// TIA Portal V17 export
// export: Created 2026-04-12T10:31:11.5882867Z, ExportSetting WithDefaults, DisplayName Totally Integrated Automation Portal, DisplayVersion V17 Update 4, DisplayName TIA Portal Openness, DisplayVersion V17 Update 4, DisplayName TIA Portal Version Control Interface, DisplayVersion V17, DisplayName SINAMICS Startdrive Advanced, DisplayVersion V17, DisplayName SINAMICS Startdrive G130, G150, S120, S150, SINAMICS MV, S210, DisplayVersion V17, DisplayName SINAMICS Startdrive G110M, G120, G120C, G120D, G120P, G115D, DisplayVersion V17, DisplayName STEP 7 Professional, DisplayVersion V17 Update 4, DisplayName STEP 7 Safety, DisplayVersion V17, DisplayName WinCC Advanced, DisplayVersion V17 Update 4
FUNCTION "PID参数控制" : Void   // FC6, LAD
{ S7_Optimized_Access := 'TRUE' }
VERSION : 0.1
// stored: AutoNumber true, IsIECCheckEnabled false, SetENOAutomatically false, UDAEnableTagReadback false
BEGIN

REGION Network 1: 采样时间
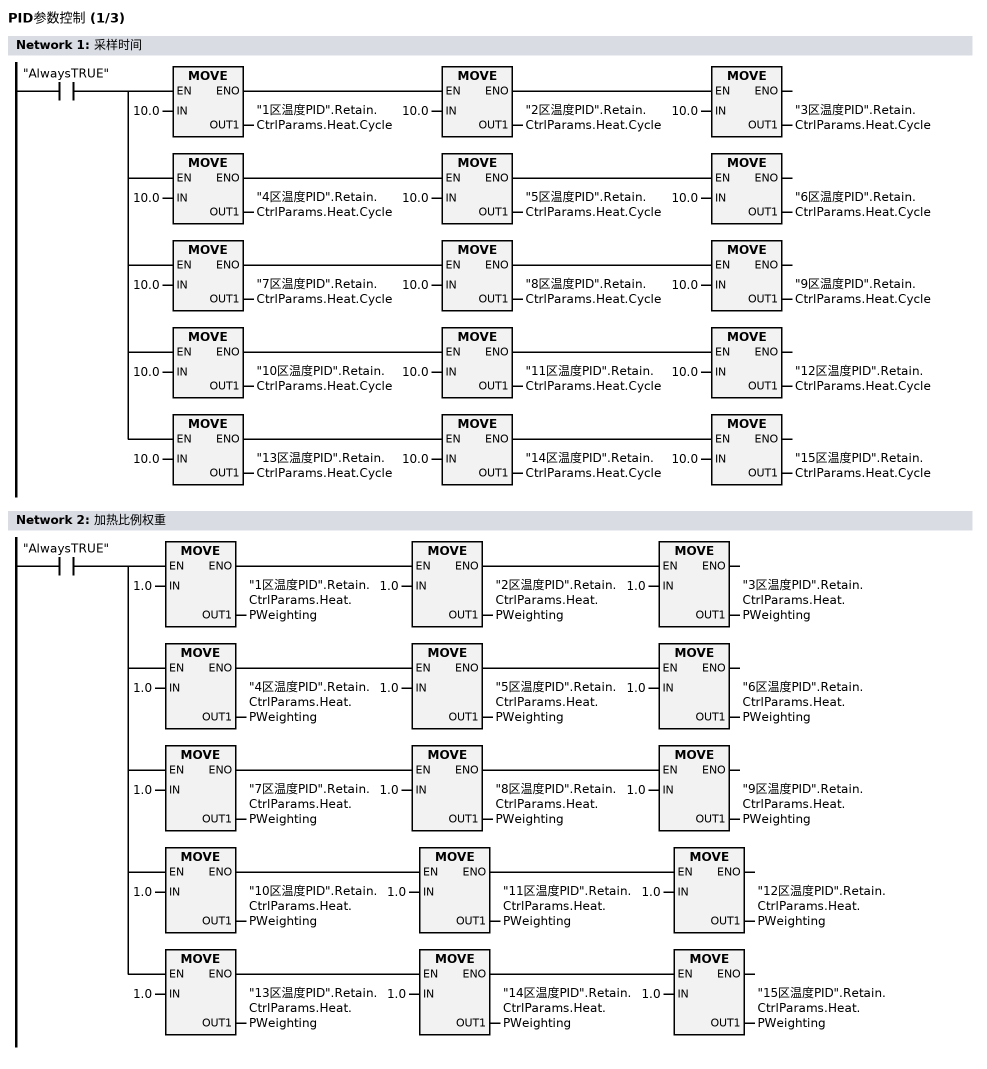
   RUNG wire#powerrail
      Contact( "AlwaysTRUE" )
      wire#w1
      Move(in := 10.0, out1 => "1区温度PID".Retain.CtrlParams.Heat.Cycle)
      Move(in := 10.0, out1 => "2区温度PID".Retain.CtrlParams.Heat.Cycle)
      Move(in := 10.0, out1 => "3区温度PID".Retain.CtrlParams.Heat.Cycle)
   END_RUNG
   RUNG wire#w1
      Move(in := 10.0, out1 => "4区温度PID".Retain.CtrlParams.Heat.Cycle)
      Move(in := 10.0, out1 => "5区温度PID".Retain.CtrlParams.Heat.Cycle)
      Move(in := 10.0, out1 => "6区温度PID".Retain.CtrlParams.Heat.Cycle)
   END_RUNG
   RUNG wire#w1
      Move(in := 10.0, out1 => "7区温度PID".Retain.CtrlParams.Heat.Cycle)
      Move(in := 10.0, out1 => "8区温度PID".Retain.CtrlParams.Heat.Cycle)
      Move(in := 10.0, out1 => "9区温度PID".Retain.CtrlParams.Heat.Cycle)
   END_RUNG
   RUNG wire#w1
      Move(in := 10.0, out1 => "10区温度PID".Retain.CtrlParams.Heat.Cycle)
      Move(in := 10.0, out1 => "11区温度PID".Retain.CtrlParams.Heat.Cycle)
      Move(in := 10.0, out1 => "12区温度PID".Retain.CtrlParams.Heat.Cycle)
   END_RUNG
   RUNG wire#w1
      Move(in := 10.0, out1 => "13区温度PID".Retain.CtrlParams.Heat.Cycle)
      Move(in := 10.0, out1 => "14区温度PID".Retain.CtrlParams.Heat.Cycle)
      Move(in := 10.0, out1 => "15区温度PID".Retain.CtrlParams.Heat.Cycle)
   END_RUNG
   // the same network as SCL:
   IF "AlwaysTRUE" THEN
       "1区温度PID".Retain.CtrlParams.Heat.Cycle := 10.0;
       "2区温度PID".Retain.CtrlParams.Heat.Cycle := 10.0;
       "3区温度PID".Retain.CtrlParams.Heat.Cycle := 10.0;
       "4区温度PID".Retain.CtrlParams.Heat.Cycle := 10.0;
       "5区温度PID".Retain.CtrlParams.Heat.Cycle := 10.0;
       "6区温度PID".Retain.CtrlParams.Heat.Cycle := 10.0;
       "7区温度PID".Retain.CtrlParams.Heat.Cycle := 10.0;
       "8区温度PID".Retain.CtrlParams.Heat.Cycle := 10.0;
       "9区温度PID".Retain.CtrlParams.Heat.Cycle := 10.0;
       "10区温度PID".Retain.CtrlParams.Heat.Cycle := 10.0;
       "11区温度PID".Retain.CtrlParams.Heat.Cycle := 10.0;
       "12区温度PID".Retain.CtrlParams.Heat.Cycle := 10.0;
       "13区温度PID".Retain.CtrlParams.Heat.Cycle := 10.0;
       "14区温度PID".Retain.CtrlParams.Heat.Cycle := 10.0;
       "15区温度PID".Retain.CtrlParams.Heat.Cycle := 10.0;
   END_IF;
END_REGION

REGION Network 2: 加热比例权重
   RUNG wire#powerrail
      Contact( "AlwaysTRUE" )
      wire#w1
      Move(in := 1.0, out1 => "1区温度PID".Retain.CtrlParams.Heat.PWeighting)
      Move(in := 1.0, out1 => "2区温度PID".Retain.CtrlParams.Heat.PWeighting)
      Move(in := 1.0, out1 => "3区温度PID".Retain.CtrlParams.Heat.PWeighting)
   END_RUNG
   RUNG wire#w1
      Move(in := 1.0, out1 => "4区温度PID".Retain.CtrlParams.Heat.PWeighting)
      Move(in := 1.0, out1 => "5区温度PID".Retain.CtrlParams.Heat.PWeighting)
      Move(in := 1.0, out1 => "6区温度PID".Retain.CtrlParams.Heat.PWeighting)
   END_RUNG
   RUNG wire#w1
      Move(in := 1.0, out1 => "7区温度PID".Retain.CtrlParams.Heat.PWeighting)
      Move(in := 1.0, out1 => "8区温度PID".Retain.CtrlParams.Heat.PWeighting)
      Move(in := 1.0, out1 => "9区温度PID".Retain.CtrlParams.Heat.PWeighting)
   END_RUNG
   RUNG wire#w1
      Move(in := 1.0, out1 => "10区温度PID".Retain.CtrlParams.Heat.PWeighting)
      Move(in := 1.0, out1 => "11区温度PID".Retain.CtrlParams.Heat.PWeighting)
      Move(in := 1.0, out1 => "12区温度PID".Retain.CtrlParams.Heat.PWeighting)
   END_RUNG
   RUNG wire#w1
      Move(in := 1.0, out1 => "13区温度PID".Retain.CtrlParams.Heat.PWeighting)
      Move(in := 1.0, out1 => "14区温度PID".Retain.CtrlParams.Heat.PWeighting)
      Move(in := 1.0, out1 => "15区温度PID".Retain.CtrlParams.Heat.PWeighting)
   END_RUNG
   // the same network as SCL:
   IF "AlwaysTRUE" THEN
       "1区温度PID".Retain.CtrlParams.Heat.PWeighting := 1.0;
       "2区温度PID".Retain.CtrlParams.Heat.PWeighting := 1.0;
       "3区温度PID".Retain.CtrlParams.Heat.PWeighting := 1.0;
       "4区温度PID".Retain.CtrlParams.Heat.PWeighting := 1.0;
       "5区温度PID".Retain.CtrlParams.Heat.PWeighting := 1.0;
       "6区温度PID".Retain.CtrlParams.Heat.PWeighting := 1.0;
       "7区温度PID".Retain.CtrlParams.Heat.PWeighting := 1.0;
       "8区温度PID".Retain.CtrlParams.Heat.PWeighting := 1.0;
       "9区温度PID".Retain.CtrlParams.Heat.PWeighting := 1.0;
       "10区温度PID".Retain.CtrlParams.Heat.PWeighting := 1.0;
       "11区温度PID".Retain.CtrlParams.Heat.PWeighting := 1.0;
       "12区温度PID".Retain.CtrlParams.Heat.PWeighting := 1.0;
       "13区温度PID".Retain.CtrlParams.Heat.PWeighting := 1.0;
       "14区温度PID".Retain.CtrlParams.Heat.PWeighting := 1.0;
       "15区温度PID".Retain.CtrlParams.Heat.PWeighting := 1.0;
   END_IF;
END_REGION

REGION Network 3: 微分比例权重
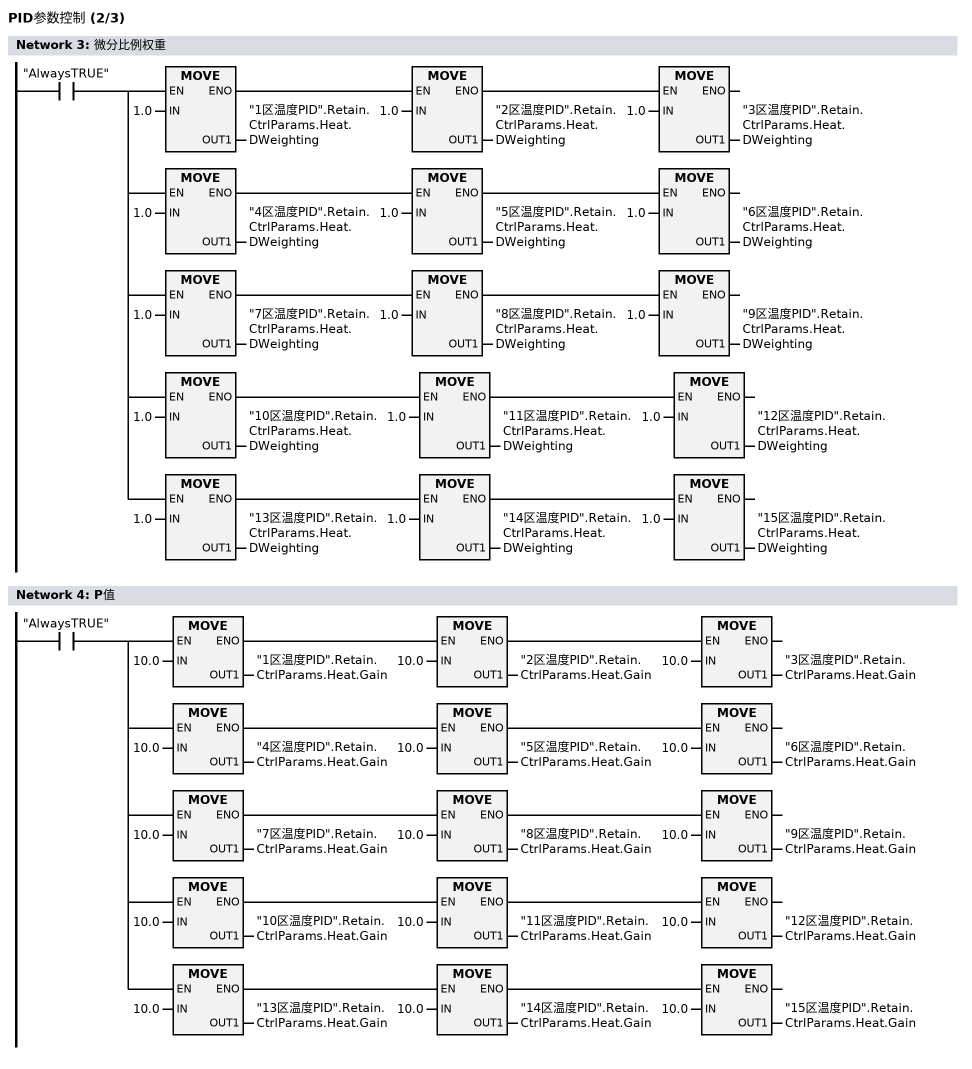
   RUNG wire#powerrail
      Contact( "AlwaysTRUE" )
      wire#w1
      Move(in := 1.0, out1 => "1区温度PID".Retain.CtrlParams.Heat.DWeighting)
      Move(in := 1.0, out1 => "2区温度PID".Retain.CtrlParams.Heat.DWeighting)
      Move(in := 1.0, out1 => "3区温度PID".Retain.CtrlParams.Heat.DWeighting)
   END_RUNG
   RUNG wire#w1
      Move(in := 1.0, out1 => "4区温度PID".Retain.CtrlParams.Heat.DWeighting)
      Move(in := 1.0, out1 => "5区温度PID".Retain.CtrlParams.Heat.DWeighting)
      Move(in := 1.0, out1 => "6区温度PID".Retain.CtrlParams.Heat.DWeighting)
   END_RUNG
   RUNG wire#w1
      Move(in := 1.0, out1 => "7区温度PID".Retain.CtrlParams.Heat.DWeighting)
      Move(in := 1.0, out1 => "8区温度PID".Retain.CtrlParams.Heat.DWeighting)
      Move(in := 1.0, out1 => "9区温度PID".Retain.CtrlParams.Heat.DWeighting)
   END_RUNG
   RUNG wire#w1
      Move(in := 1.0, out1 => "10区温度PID".Retain.CtrlParams.Heat.DWeighting)
      Move(in := 1.0, out1 => "11区温度PID".Retain.CtrlParams.Heat.DWeighting)
      Move(in := 1.0, out1 => "12区温度PID".Retain.CtrlParams.Heat.DWeighting)
   END_RUNG
   RUNG wire#w1
      Move(in := 1.0, out1 => "13区温度PID".Retain.CtrlParams.Heat.DWeighting)
      Move(in := 1.0, out1 => "14区温度PID".Retain.CtrlParams.Heat.DWeighting)
      Move(in := 1.0, out1 => "15区温度PID".Retain.CtrlParams.Heat.DWeighting)
   END_RUNG
   // the same network as SCL:
   IF "AlwaysTRUE" THEN
       "1区温度PID".Retain.CtrlParams.Heat.DWeighting := 1.0;
       "2区温度PID".Retain.CtrlParams.Heat.DWeighting := 1.0;
       "3区温度PID".Retain.CtrlParams.Heat.DWeighting := 1.0;
       "4区温度PID".Retain.CtrlParams.Heat.DWeighting := 1.0;
       "5区温度PID".Retain.CtrlParams.Heat.DWeighting := 1.0;
       "6区温度PID".Retain.CtrlParams.Heat.DWeighting := 1.0;
       "7区温度PID".Retain.CtrlParams.Heat.DWeighting := 1.0;
       "8区温度PID".Retain.CtrlParams.Heat.DWeighting := 1.0;
       "9区温度PID".Retain.CtrlParams.Heat.DWeighting := 1.0;
       "10区温度PID".Retain.CtrlParams.Heat.DWeighting := 1.0;
       "11区温度PID".Retain.CtrlParams.Heat.DWeighting := 1.0;
       "12区温度PID".Retain.CtrlParams.Heat.DWeighting := 1.0;
       "13区温度PID".Retain.CtrlParams.Heat.DWeighting := 1.0;
       "14区温度PID".Retain.CtrlParams.Heat.DWeighting := 1.0;
       "15区温度PID".Retain.CtrlParams.Heat.DWeighting := 1.0;
   END_IF;
END_REGION

REGION Network 4: P值
   RUNG wire#powerrail
      Contact( "AlwaysTRUE" )
      wire#w1
      Move(in := 10.0, out1 => "1区温度PID".Retain.CtrlParams.Heat.Gain)
      Move(in := 10.0, out1 => "2区温度PID".Retain.CtrlParams.Heat.Gain)
      Move(in := 10.0, out1 => "3区温度PID".Retain.CtrlParams.Heat.Gain)
   END_RUNG
   RUNG wire#w1
      Move(in := 10.0, out1 => "4区温度PID".Retain.CtrlParams.Heat.Gain)
      Move(in := 10.0, out1 => "5区温度PID".Retain.CtrlParams.Heat.Gain)
      Move(in := 10.0, out1 => "6区温度PID".Retain.CtrlParams.Heat.Gain)
   END_RUNG
   RUNG wire#w1
      Move(in := 10.0, out1 => "7区温度PID".Retain.CtrlParams.Heat.Gain)
      Move(in := 10.0, out1 => "8区温度PID".Retain.CtrlParams.Heat.Gain)
      Move(in := 10.0, out1 => "9区温度PID".Retain.CtrlParams.Heat.Gain)
   END_RUNG
   RUNG wire#w1
      Move(in := 10.0, out1 => "10区温度PID".Retain.CtrlParams.Heat.Gain)
      Move(in := 10.0, out1 => "11区温度PID".Retain.CtrlParams.Heat.Gain)
      Move(in := 10.0, out1 => "12区温度PID".Retain.CtrlParams.Heat.Gain)
   END_RUNG
   RUNG wire#w1
      Move(in := 10.0, out1 => "13区温度PID".Retain.CtrlParams.Heat.Gain)
      Move(in := 10.0, out1 => "14区温度PID".Retain.CtrlParams.Heat.Gain)
      Move(in := 10.0, out1 => "15区温度PID".Retain.CtrlParams.Heat.Gain)
   END_RUNG
   // the same network as SCL:
   IF "AlwaysTRUE" THEN
       "1区温度PID".Retain.CtrlParams.Heat.Gain := 10.0;
       "2区温度PID".Retain.CtrlParams.Heat.Gain := 10.0;
       "3区温度PID".Retain.CtrlParams.Heat.Gain := 10.0;
       "4区温度PID".Retain.CtrlParams.Heat.Gain := 10.0;
       "5区温度PID".Retain.CtrlParams.Heat.Gain := 10.0;
       "6区温度PID".Retain.CtrlParams.Heat.Gain := 10.0;
       "7区温度PID".Retain.CtrlParams.Heat.Gain := 10.0;
       "8区温度PID".Retain.CtrlParams.Heat.Gain := 10.0;
       "9区温度PID".Retain.CtrlParams.Heat.Gain := 10.0;
       "10区温度PID".Retain.CtrlParams.Heat.Gain := 10.0;
       "11区温度PID".Retain.CtrlParams.Heat.Gain := 10.0;
       "12区温度PID".Retain.CtrlParams.Heat.Gain := 10.0;
       "13区温度PID".Retain.CtrlParams.Heat.Gain := 10.0;
       "14区温度PID".Retain.CtrlParams.Heat.Gain := 10.0;
       "15区温度PID".Retain.CtrlParams.Heat.Gain := 10.0;
   END_IF;
END_REGION

REGION Network 5: I值
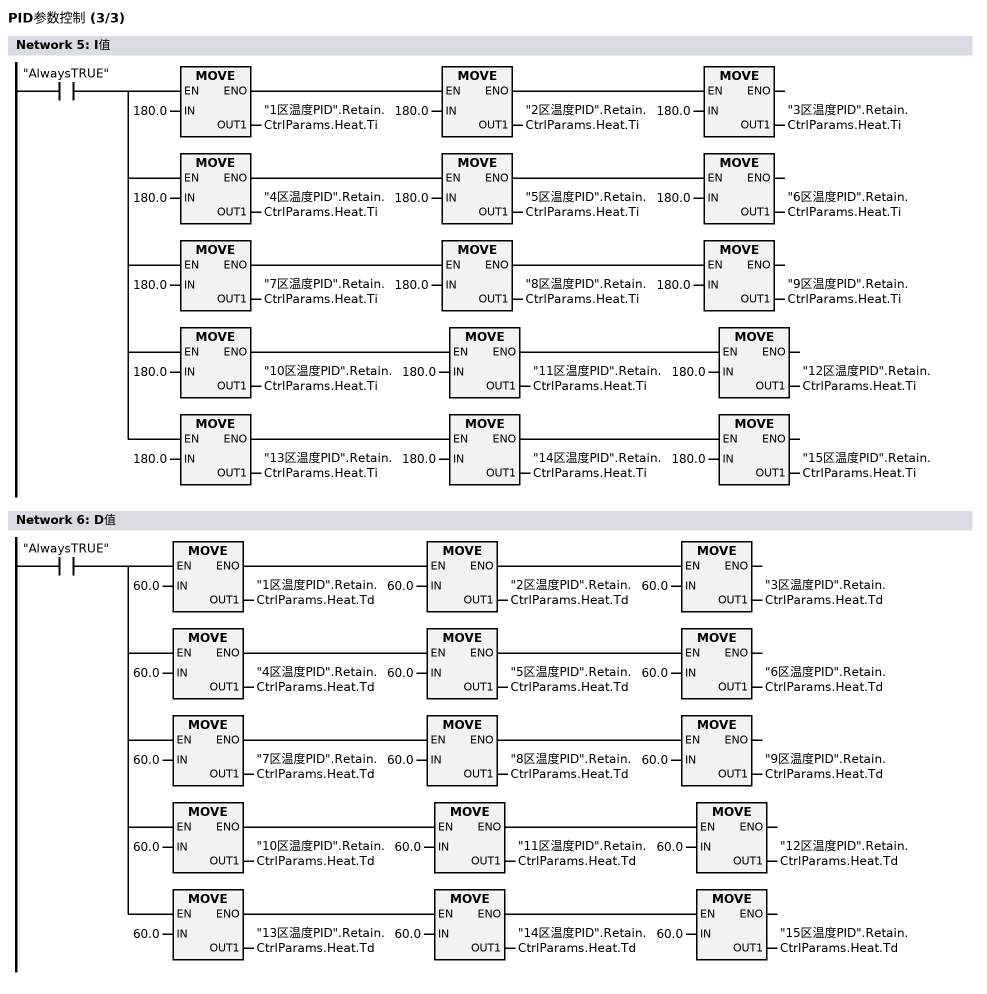
   RUNG wire#powerrail
      Contact( "AlwaysTRUE" )
      wire#w1
      Move(in := 180.0, out1 => "1区温度PID".Retain.CtrlParams.Heat.Ti)
      Move(in := 180.0, out1 => "2区温度PID".Retain.CtrlParams.Heat.Ti)
      Move(in := 180.0, out1 => "3区温度PID".Retain.CtrlParams.Heat.Ti)
   END_RUNG
   RUNG wire#w1
      Move(in := 180.0, out1 => "4区温度PID".Retain.CtrlParams.Heat.Ti)
      Move(in := 180.0, out1 => "5区温度PID".Retain.CtrlParams.Heat.Ti)
      Move(in := 180.0, out1 => "6区温度PID".Retain.CtrlParams.Heat.Ti)
   END_RUNG
   RUNG wire#w1
      Move(in := 180.0, out1 => "7区温度PID".Retain.CtrlParams.Heat.Ti)
      Move(in := 180.0, out1 => "8区温度PID".Retain.CtrlParams.Heat.Ti)
      Move(in := 180.0, out1 => "9区温度PID".Retain.CtrlParams.Heat.Ti)
   END_RUNG
   RUNG wire#w1
      Move(in := 180.0, out1 => "10区温度PID".Retain.CtrlParams.Heat.Ti)
      Move(in := 180.0, out1 => "11区温度PID".Retain.CtrlParams.Heat.Ti)
      Move(in := 180.0, out1 => "12区温度PID".Retain.CtrlParams.Heat.Ti)
   END_RUNG
   RUNG wire#w1
      Move(in := 180.0, out1 => "13区温度PID".Retain.CtrlParams.Heat.Ti)
      Move(in := 180.0, out1 => "14区温度PID".Retain.CtrlParams.Heat.Ti)
      Move(in := 180.0, out1 => "15区温度PID".Retain.CtrlParams.Heat.Ti)
   END_RUNG
   // the same network as SCL:
   IF "AlwaysTRUE" THEN
       "1区温度PID".Retain.CtrlParams.Heat.Ti := 180.0;
       "2区温度PID".Retain.CtrlParams.Heat.Ti := 180.0;
       "3区温度PID".Retain.CtrlParams.Heat.Ti := 180.0;
       "4区温度PID".Retain.CtrlParams.Heat.Ti := 180.0;
       "5区温度PID".Retain.CtrlParams.Heat.Ti := 180.0;
       "6区温度PID".Retain.CtrlParams.Heat.Ti := 180.0;
       "7区温度PID".Retain.CtrlParams.Heat.Ti := 180.0;
       "8区温度PID".Retain.CtrlParams.Heat.Ti := 180.0;
       "9区温度PID".Retain.CtrlParams.Heat.Ti := 180.0;
       "10区温度PID".Retain.CtrlParams.Heat.Ti := 180.0;
       "11区温度PID".Retain.CtrlParams.Heat.Ti := 180.0;
       "12区温度PID".Retain.CtrlParams.Heat.Ti := 180.0;
       "13区温度PID".Retain.CtrlParams.Heat.Ti := 180.0;
       "14区温度PID".Retain.CtrlParams.Heat.Ti := 180.0;
       "15区温度PID".Retain.CtrlParams.Heat.Ti := 180.0;
   END_IF;
END_REGION

REGION Network 6: D值
   RUNG wire#powerrail
      Contact( "AlwaysTRUE" )
      wire#w1
      Move(in := 60.0, out1 => "1区温度PID".Retain.CtrlParams.Heat.Td)
      Move(in := 60.0, out1 => "2区温度PID".Retain.CtrlParams.Heat.Td)
      Move(in := 60.0, out1 => "3区温度PID".Retain.CtrlParams.Heat.Td)
   END_RUNG
   RUNG wire#w1
      Move(in := 60.0, out1 => "4区温度PID".Retain.CtrlParams.Heat.Td)
      Move(in := 60.0, out1 => "5区温度PID".Retain.CtrlParams.Heat.Td)
      Move(in := 60.0, out1 => "6区温度PID".Retain.CtrlParams.Heat.Td)
   END_RUNG
   RUNG wire#w1
      Move(in := 60.0, out1 => "7区温度PID".Retain.CtrlParams.Heat.Td)
      Move(in := 60.0, out1 => "8区温度PID".Retain.CtrlParams.Heat.Td)
      Move(in := 60.0, out1 => "9区温度PID".Retain.CtrlParams.Heat.Td)
   END_RUNG
   RUNG wire#w1
      Move(in := 60.0, out1 => "10区温度PID".Retain.CtrlParams.Heat.Td)
      Move(in := 60.0, out1 => "11区温度PID".Retain.CtrlParams.Heat.Td)
      Move(in := 60.0, out1 => "12区温度PID".Retain.CtrlParams.Heat.Td)
   END_RUNG
   RUNG wire#w1
      Move(in := 60.0, out1 => "13区温度PID".Retain.CtrlParams.Heat.Td)
      Move(in := 60.0, out1 => "14区温度PID".Retain.CtrlParams.Heat.Td)
      Move(in := 60.0, out1 => "15区温度PID".Retain.CtrlParams.Heat.Td)
   END_RUNG
   // the same network as SCL:
   IF "AlwaysTRUE" THEN
       "1区温度PID".Retain.CtrlParams.Heat.Td := 60.0;
       "2区温度PID".Retain.CtrlParams.Heat.Td := 60.0;
       "3区温度PID".Retain.CtrlParams.Heat.Td := 60.0;
       "4区温度PID".Retain.CtrlParams.Heat.Td := 60.0;
       "5区温度PID".Retain.CtrlParams.Heat.Td := 60.0;
       "6区温度PID".Retain.CtrlParams.Heat.Td := 60.0;
       "7区温度PID".Retain.CtrlParams.Heat.Td := 60.0;
       "8区温度PID".Retain.CtrlParams.Heat.Td := 60.0;
       "9区温度PID".Retain.CtrlParams.Heat.Td := 60.0;
       "10区温度PID".Retain.CtrlParams.Heat.Td := 60.0;
       "11区温度PID".Retain.CtrlParams.Heat.Td := 60.0;
       "12区温度PID".Retain.CtrlParams.Heat.Td := 60.0;
       "13区温度PID".Retain.CtrlParams.Heat.Td := 60.0;
       "14区温度PID".Retain.CtrlParams.Heat.Td := 60.0;
       "15区温度PID".Retain.CtrlParams.Heat.Td := 60.0;
   END_IF;
END_REGION
END_FUNCTION
